TYPE ST_EL5042_Status :
STRUCT
END_STRUCT
END_TYPE

(* stored: Version 1.1.0.1
   DUT ST_EL5042_Status: Id {fe0ff67d-e11f-4b59-99eb-dd372e356d77} *)
